INTERFACE I_State EXTENDS I_Tagged, I_Debug, I_StateAdapter

PROPERTY Owner : I_Entity
GET
END_GET
END_PROPERTY

END_INTERFACE

(* stored: Version 1.1.0.1
   Itf I_State: Id {8ee68e54-e03a-40c4-b9fd-28674c83f71b}
   Property Owner: Id {0bc823ea-d1a3-4234-8eb6-66bbb0f8e330}
   Get Get: Id {5525b7b9-1d3e-4516-9f77-c77dffb34dd8} *)
